// SIMATIC S7-200 SMART project (STEP 7-Micro/WIN SMART), CPU SR40

SYMBOL_TABLE 系统符号
Clock_1s         SM0.5    // 针对 1 s 的周期时间，时钟脉冲接通 0.5 s，断开 0.5 s.
END_SYMBOL_TABLE

ORGANIZATION_BLOCK MAIN:OB1
TITLE=程序注释
BEGIN
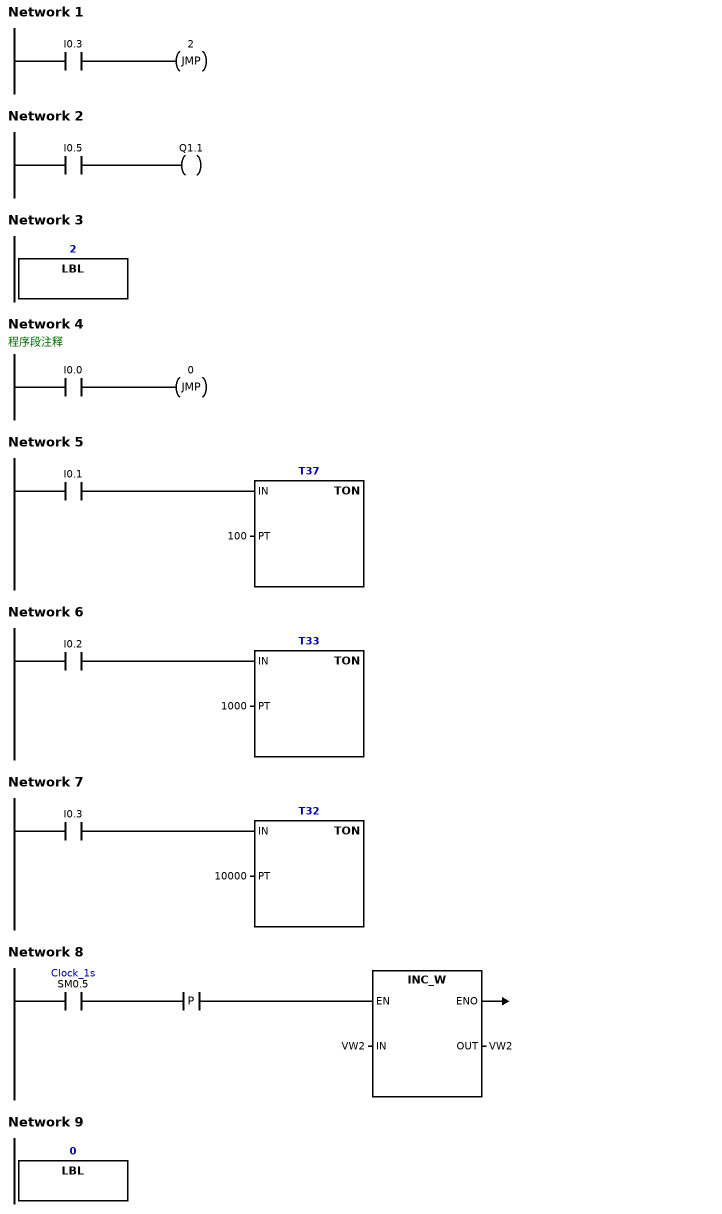
Network 1
LD     I0.3
JMP    2
Network 2
LD     I0.5
=      Q1.1
Network 3
LBL    2
Network 4
// 程序段注释
// I0.0为1状态时跳转条件满足
LD     I0.0
JMP    0
Network 5
// 100ms定时器，设定值为10s
LD     I0.1
TON    T37, 100
Network 6
// 10ms定时器，设定值为10s
LD     I0.2
TON    T33, 1000
Network 7
// 1ms定时器，设定值为10s
LD     I0.3
TON    T32, 10000
Network 8
LD     Clock_1s:SM0.5
EU
INCW   VW2
Network 9
LBL    0
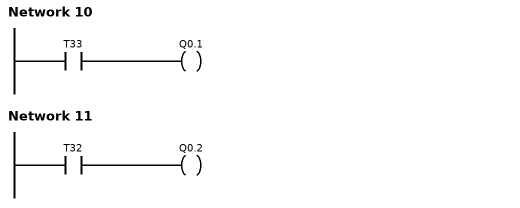
Network 10
LD     T33
=      Q0.1
Network 11
LD     T32
=      Q0.2
END_ORGANIZATION_BLOCK
